{attribute addProperty BoxType "EL3483-0060-0018"}
{attribute addProperty Id "L1_StatusAT %I*L1_Status_2BC7A2034050L1_BasicAT %I*L1_Basic_FE52C16D3240L2_StatusAT %I*L2_Status_2BC7A2034050L2_BasicAT %I*L2_Basic_FE52C16D3240L3_StatusAT %I*L3_Status_2BC7A2034050L3_BasicAT %I*L3_Basic_FE52C16D3240Total_StatusAT %I*Total_Status_5266C05996120Total_AdvancedAT %I*Total_Advanced_FCA492E91620Total_Total_L_L_VoltageAT %I*Total_Total_L_L_Voltage_36E7ACB196120WcStateAT %I*WcState_98A4DF7520.250InfoDataAT %I*InfoData_BC63D37F80100"}
{attribute addProperty CRC "1757155362"}
{attribute addProperty SizeInBites "506"}
{attribute addProperty SizeInBytes "63.25"}
TYPE EL3483_2724D368 :
STRUCT
	{attribute addProperty Name "L1_Status"}
	L1_Status : L1_Status_2BC7A203;
	{attribute addProperty Name "L1_Basic"}
	L1_Basic : L1_Basic_FE52C16D;
	{attribute addProperty Name "L2_Status"}
	L2_Status : L2_Status_2BC7A203;
	{attribute addProperty Name "L2_Basic"}
	L2_Basic : L2_Basic_FE52C16D;
	{attribute addProperty Name "L3_Status"}
	L3_Status : L3_Status_2BC7A203;
	{attribute addProperty Name "L3_Basic"}
	L3_Basic : L3_Basic_FE52C16D;
	{attribute addProperty Name "Total_Status"}
	Total_Status : Total_Status_5266C059;
	{attribute addProperty Name "Total_Advanced"}
	Total_Advanced : Total_Advanced_FCA492E9;
	{attribute addProperty Name "Total_Total_L_L_Voltage"}
	Total_Total_L_L_Voltage : Total_Total_L_L_Voltage_36E7ACB1;
	{attribute addProperty Name "WcState"}
	WcState : WcState_98A4DF75;
	{attribute addProperty Name "InfoData"}
	InfoData : InfoData_BC63D37F;
END_STRUCT
END_TYPE

(* stored: Version 1.2.0.0, ProductVersion 3.1.4024.9
   DUT EL3483_2724D368: Id {a8bea8de-adac-4da0-84a2-73462b3a6d13} *)
